FUNCTION_BLOCK CoeDevice EXTENDS CyclicComponent IMPLEMENTS I_CoeDevice, I_CoeTransfer
VAR
	{attribute 'hide'}
	_Error : BOOL;
	{attribute 'hide'}
	_Busy : BOOL;
	{attribute 'hide'}
	_ErrorId : UDINT;
	{attribute 'hide'}
	_ActiveIsWrite : BOOL;
	_AdsAddr   : REFERENCE TO AMSADDR;
	_Scheduler : I_CoeTransferScheduler; // optional: services this device while a transfer is in flight
	CoeRead	   : FB_EcCoESdoReadEx;
	CoeWrite   : FB_EcCoESdoWriteEx;
END_VAR

VAR CONSTANT
	ERROR_NO_ADDRESS : UDINT := 16#70B; // ADS: invalid parameter - AdsAddr reference not set
END_VAR

PROPERTY AdsAddr : REFERENCE TO AMSADDR
GET
AdsAddr REF= _AdsAddr;
END_GET
SET
_AdsAddr REF= AdsAddr;
END_SET
END_PROPERTY

{attribute 'monitoring' := 'call'}
PROPERTY Busy : BOOL
GET
Busy := _Busy;
END_GET
END_PROPERTY

// Services the SDO transfer in flight. Call each cycle while Busy; with a Scheduler set the
// scheduler does this for you.
METHOD CyclicLogic
VAR_INST
END_VAR
IF NOT __ISVALIDREF(_AdsAddr) THEN
	RETURN;
END_IF

CoeRead(sNetId := F_CreateAmsNetId(_AdsAddr.netId), nSlaveAddr := _AdsAddr.port, tTimeout := T#1S);
CoeWrite(sNetId := F_CreateAmsNetId(_AdsAddr.netId), nSlaveAddr := _AdsAddr.port, tTimeout := T#1S);
CoeRead.bExecute  := FALSE;
CoeWrite.bExecute := FALSE;

(* Only the active function block decides Busy/Error: a stale bError of the other one must not leak. *)
IF _ActiveIsWrite THEN
	_Busy := CoeWrite.bBusy;
	IF CoeWrite.bError THEN
		_Error	 := TRUE;
		_ErrorId := CoeWrite.nErrId;
	END_IF
ELSE
	_Busy := CoeRead.bBusy;
	IF CoeRead.bError THEN
		_Error	 := TRUE;
		_ErrorId := CoeRead.nErrId;
	END_IF
END_IF
END_METHOD

{attribute 'monitoring' := 'call'}
PROPERTY Error : BOOL
GET
Error := _Error;
END_GET
END_PROPERTY

{attribute 'monitoring' := 'call'}
PROPERTY ErrorId : UDINT
GET
ErrorID := _ErrorID;
END_GET
END_PROPERTY

// Starts an SDO read; ignored while Busy. Fails with ERROR_NO_ADDRESS if AdsAddr is not set.
METHOD Read
VAR_INPUT
	Index	 : WORD;
	SubIndex : BYTE;
	pDstBuf	 : PVOID;
	BufLen	 : UDINT;
END_VAR
IF _Busy THEN
	RETURN;
END_IF

IF NOT __ISVALIDREF(_AdsAddr) THEN
	_Error	 := TRUE;
	_ErrorId := ERROR_NO_ADDRESS;
	RETURN;
END_IF

CoeRead.nSubIndex		:= SubIndex;
CoeRead.nIndex			:= Index;
CoeRead.pDstBuf			:= pDstBuf;
CoeRead.cbBufLen		:= BufLen;
CoeRead.bCompleteAccess := SubIndex = 0;
_ActiveIsWrite			:= FALSE;
_Error					:= FALSE;
_ErrorId				:= 0;
_Busy					:= TRUE;
CoeRead.bExecute		:= TRUE;

IF _Scheduler <> 0 THEN
	_Scheduler.Register(THIS^);
END_IF
END_METHOD

// Optional scheduler that calls CyclicLogic while a transfer is in flight (set by EtherCatIoDevice).
PROPERTY Scheduler : I_CoeTransferScheduler
GET
Scheduler := _Scheduler;
END_GET
SET
_Scheduler := Scheduler;
END_SET
END_PROPERTY

// Starts an SDO write from pDstBuf (used as the source buffer); ignored while Busy.
METHOD Write
VAR_INPUT
	Index	 : WORD;
	SubIndex : BYTE;
	pDstBuf	 : PVOID;
	BufLen	 : UDINT;
END_VAR
IF _Busy THEN
	RETURN;
END_IF

IF NOT __ISVALIDREF(_AdsAddr) THEN
	_Error	 := TRUE;
	_ErrorId := ERROR_NO_ADDRESS;
	RETURN;
END_IF

CoeWrite.nSubIndex		 := SubIndex;
CoeWrite.nIndex			 := Index;
CoeWrite.pSrcBuf		 := pDstBuf;
CoeWrite.cbBufLen		 := BufLen;
CoeWrite.bCompleteAccess := SubIndex = 0;
_ActiveIsWrite			 := TRUE;
_Error					 := FALSE;
_ErrorId				 := 0;
_Busy					 := TRUE;
CoeWrite.bExecute		 := TRUE;

IF _Scheduler <> 0 THEN
	_Scheduler.Register(THIS^);
END_IF
END_METHOD

END_FUNCTION_BLOCK

(* stored: Version 1.1.0.1, ProductVersion 3.1.4026.18
   POU CoeDevice: Id {c44fc925-b48d-43e7-9921-59d1275857d3}, SpecialFunc None
   Folder TaskResult: Id {f08d9870-c876-4e92-a979-edd7606478ba}
   Property AdsAddr: Id {809820b6-2843-4b61-8ee7-e554a700fe77}
   Get Get: Id {791cbbcb-db0a-402b-b1c3-3fd5592e95c8}
   Set Set: Id {b5264c88-f20b-45c4-bbe2-a7789a6ce714}
   Property Busy: Id {662175c3-e675-4259-997a-bb32092b5b95}
   Get Get: Id {7d0a2fa5-2cb6-4a1f-91d9-341a496cb410}
   Method CyclicLogic: Id {f7dc4c56-720e-4dcf-a90e-1437f6929992}
   Property Error: Id {06a86ac8-f65a-409c-a4f6-bbee7cc5c268}
   Get Get: Id {bda23b4a-c206-4d73-9042-d2dd16e3532a}
   Property ErrorId: Id {a6c4d22e-d553-43cc-9f33-712949103b8a}
   Get Get: Id {5bc44fad-a426-4789-b7d0-b9ee3f9a3787}
   Method Read: Id {d76200df-b7b1-4642-b3bc-ba548d1d54d4}
   Property Scheduler: Id {7446c31d-3cf4-4065-bce9-980d3c94b960}
   Get Get: Id {4b6a3fca-f994-47db-b71b-7fdbbdccd5ed}
   Set Set: Id {6a20a12b-649e-4f0c-bee0-f85b238f9c3c}
   Method Write: Id {f028f408-1739-4375-a0d7-b0a99ab310d9} *)
